(* Schneider Machine Expert - Basic project Grafcet con botonera y flotantes, file version 2.7.0.0 *)
(* ProjectInformations: Name=Nuevo proyecto *)

HARDWARE
  Cpu 0: TM221M16R/G
  ModuleExtensionObject 0: TM3DI16K
  ModuleExtensionObject 1: TM3AI4/G
  EthernetConfiguration: NetworkName=M221, IpAllocationMode=FixedAddress, IpAddress=0.0.0.0, SubnetMask=0.0.0.0
  SerialLineConfiguration: Baud=Baud19200, Parity=ParityEven, DataBits=DataBits8, StopBits=StopBits1, PhysicalMedium=PhysicalMediumRs485, TransmissionMode=TransmissionModeModbusRtu, SlaveId=1, Addressing=SlaveAddressing
  MastTask: UsePeriodScanMode=false, PeriodScan=100
  FastTask: Period=255
  CpuBehavior: StartingMode=StartAsPreviousState, AutoSaveRamOnEeprom=true, WatchdogPeriod=250

SYMBOLS  (address, symbol, comment, settings)
  %M0         "Item detected"
  %M1         "Lid at place"
  %M2         "Base at place"
  %M3         "Part leaving"
  %M4         "Start"
  %M5         "Reset"
  %M6         "Stop"
  %M8         "Auto"
  %M10        "Lids conveyor 1"
  %M11        "Stop blade 1"
  %M13        "Base conveyor 1"
  %M14        "Stop blade 2"
  %M15        "Bases conveyor 2"
  %M16        "Grab"
  %M17        "Start light"
  %M18        "Rest light"
  %M19        "Stop light"
  %M100       "Encendido"
  %X2         "Estado 2"
  %X3         "Estado 3"
  %X5         "Estado 5"
  %X6         "Estado 6"
  %X7         "Estado 7"
  %X8         "Estado 8"
  %X9         "Estado 9"
  %X11        "Estado 11"
  %TM0        "Temporizador estado 11"  [Preset=9, Base=OneSecond]
  %C0         "Contador de piezas finalizadas"  [Preset=1000]

GRAFCET Grafcet Secundario
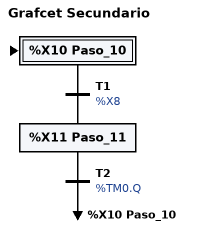
  INITIAL_STEP %X10  (* Paso_10 *)
  STEP %X11  (* Paso_11 *)
  TRANSITION T1 FROM %X10 TO %X11 := %X8;
  TRANSITION T2 FROM %X11 TO %X10 := %TM0.Q;

GRAFCET Grafcet Principal
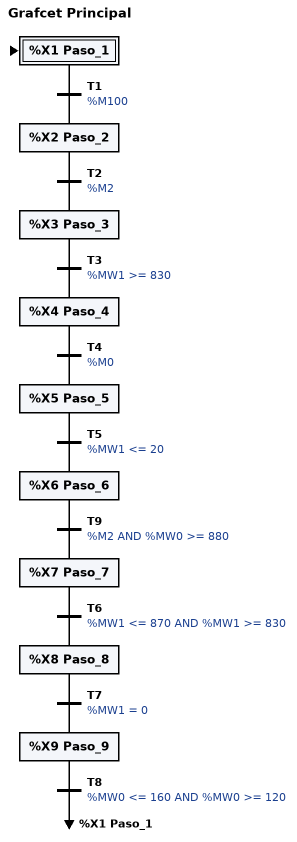
  INITIAL_STEP %X1  (* Paso_1 *)
  STEP %X2  (* Paso_2 *)
  STEP %X3  (* Paso_3 *)
  STEP %X4  (* Paso_4 *)
  STEP %X5  (* Paso_5 *)
  STEP %X6  (* Paso_6 *)
  STEP %X7  (* Paso_7 *)
  STEP %X8  (* Paso_8 *)
  STEP %X9  (* Paso_9 *)
  TRANSITION T1 FROM %X1 TO %X2 := %M100;
  TRANSITION T2 FROM %X2 TO %X3 := %M2;
  TRANSITION T3 FROM %X3 TO %X4 := %MW1 >= 830;
  TRANSITION T4 FROM %X4 TO %X5 := %M0;
  TRANSITION T5 FROM %X5 TO %X6 := %MW1 <= 20;
  TRANSITION T6 FROM %X7 TO %X8 := %MW1 <= 870 AND %MW1 >= 830;
  TRANSITION T7 FROM %X8 TO %X9 := %MW1 = 0;
  TRANSITION T8 FROM %X9 TO %X1 := %MW0 <= 160 AND %MW0 >= 120;
  TRANSITION T9 FROM %X6 TO %X7 := %M2 AND %MW0 >= 880;

TRANSITION T1 (%X10 -> %X11) 
  (* SectionNumber=0 *)

// Rung 0: Tr1
  LD %X8
  ENDT
  // as ST:
  //   TRANSITION := %X8;

TRANSITION T2 (%X11 -> %X10) 
  (* SectionNumber=0 *)

// Rung 1: Tr2
  LD %TM0.Q
  ENDT
  // as ST:
  //   TRANSITION := %TM0.Q;

TRANSITION T1 (%X1 -> %X2) 
  (* SectionNumber=0 *)

// Rung 2: Tr1
  LD %M100
  ENDT
  // as ST:
  //   TRANSITION := %M100;

TRANSITION T2 (%X2 -> %X3) 
  (* SectionNumber=0 *)

// Rung 3: Tr2
  LD %M2
  ENDT
  // as ST:
  //   TRANSITION := %M2;

TRANSITION T3 (%X3 -> %X4) 
  (* SectionNumber=0 *)

// Rung 4: Tr3
  LD [ %MW1 >= 830 ]
  ENDT
  // as ST:
  //   TRANSITION := %MW1 >= 830;

TRANSITION T4 (%X4 -> %X5) 
  (* SectionNumber=0 *)

// Rung 5: Tr4
  LD %M0
  ENDT
  // as ST:
  //   TRANSITION := %M0;

TRANSITION T5 (%X5 -> %X6) 
  (* SectionNumber=0 *)

// Rung 6: Tr5
  LD [ %MW1 <= 20 ]
  ENDT
  // as ST:
  //   TRANSITION := %MW1 <= 20;

TRANSITION T6 (%X7 -> %X8) 
  (* SectionNumber=0 *)

// Rung 7: Tr7
  LD [ %MW1 <= 870 ]
  AND [ %MW1 >= 830 ]
  ENDT
  // as ST:
  //   TRANSITION := %MW1 <= 870 AND %MW1 >= 830;

TRANSITION T7 (%X8 -> %X9) 
  (* SectionNumber=0 *)

// Rung 8: Tr8
  LD [ %MW1 = 0 ]
  ENDT
  // as ST:
  //   TRANSITION := %MW1 = 0;

TRANSITION T8 (%X9 -> %X1) 
  (* SectionNumber=0 *)

// Rung 9: Tr9
  LD [ %MW0 <= 160 ]
  AND [ %MW0 >= 120 ]
  ENDT
  // as ST:
  //   TRANSITION := %MW0 <= 160 AND %MW0 >= 120;

TRANSITION T9 (%X6 -> %X7) 
  (* SectionNumber=0 *)

// Rung 10: Tr6
  LD %M2
  AND [ %MW0 >= 880 ]
  ENDT
  // as ST:
  //   TRANSITION := %M2 AND %MW0 >= 880;

POU Botonera
  (* SectionNumber=13 *)

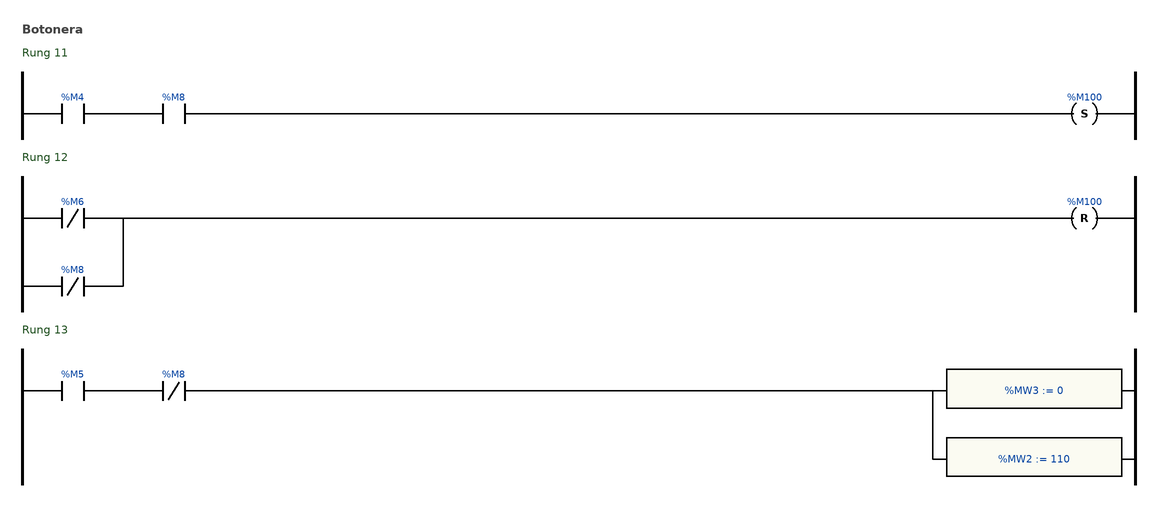

// Rung 11
  LD %M4
  AND %M8
  S %M100
  // as ST:
  //   IF %M4 AND %M8 THEN %M100 := TRUE; END_IF;

// Rung 12
  LDN %M6
  ORN %M8
  R %M100
  // as ST:
  //   IF NOT %M6 OR NOT %M8 THEN %M100 := FALSE; END_IF;

// Rung 13
  LD %M5
  ANDN %M8
  [ %MW3 := 0 ]
  [ %MW2 := 110 ]
  // as ST:
  //   IF %M5 AND NOT %M8 THEN %MW3 := 0; END_IF;
  //   IF %M5 AND NOT %M8 THEN %MW2 := 110; END_IF;

POU Pilotos
  (* SectionNumber=14 *)

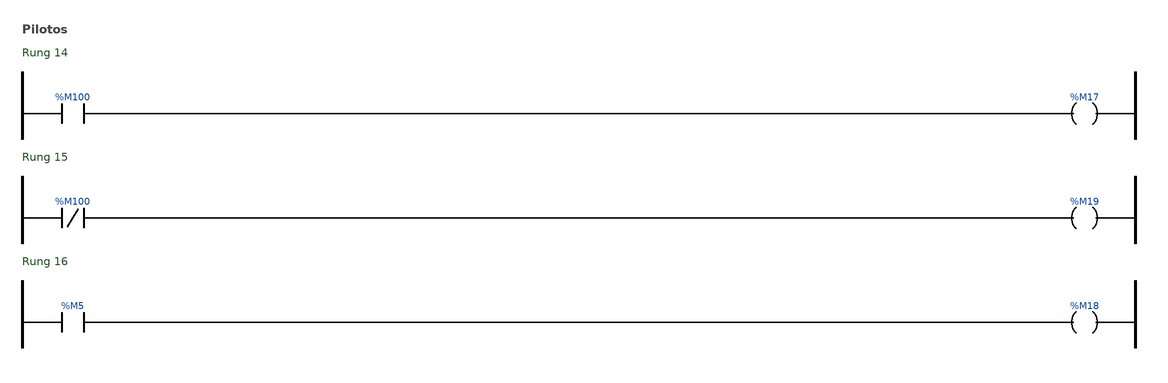

// Rung 14
  LD %M100
  ST %M17
  // as ST:
  //   %M17 := %M100;

// Rung 15
  LDN %M100
  ST %M19
  // as ST:
  //   %M19 := NOT %M100;

// Rung 16
  LD %M5
  ST %M18
  // as ST:
  //   %M18 := %M5;

POU Acciones
  (* SectionNumber=15 *)

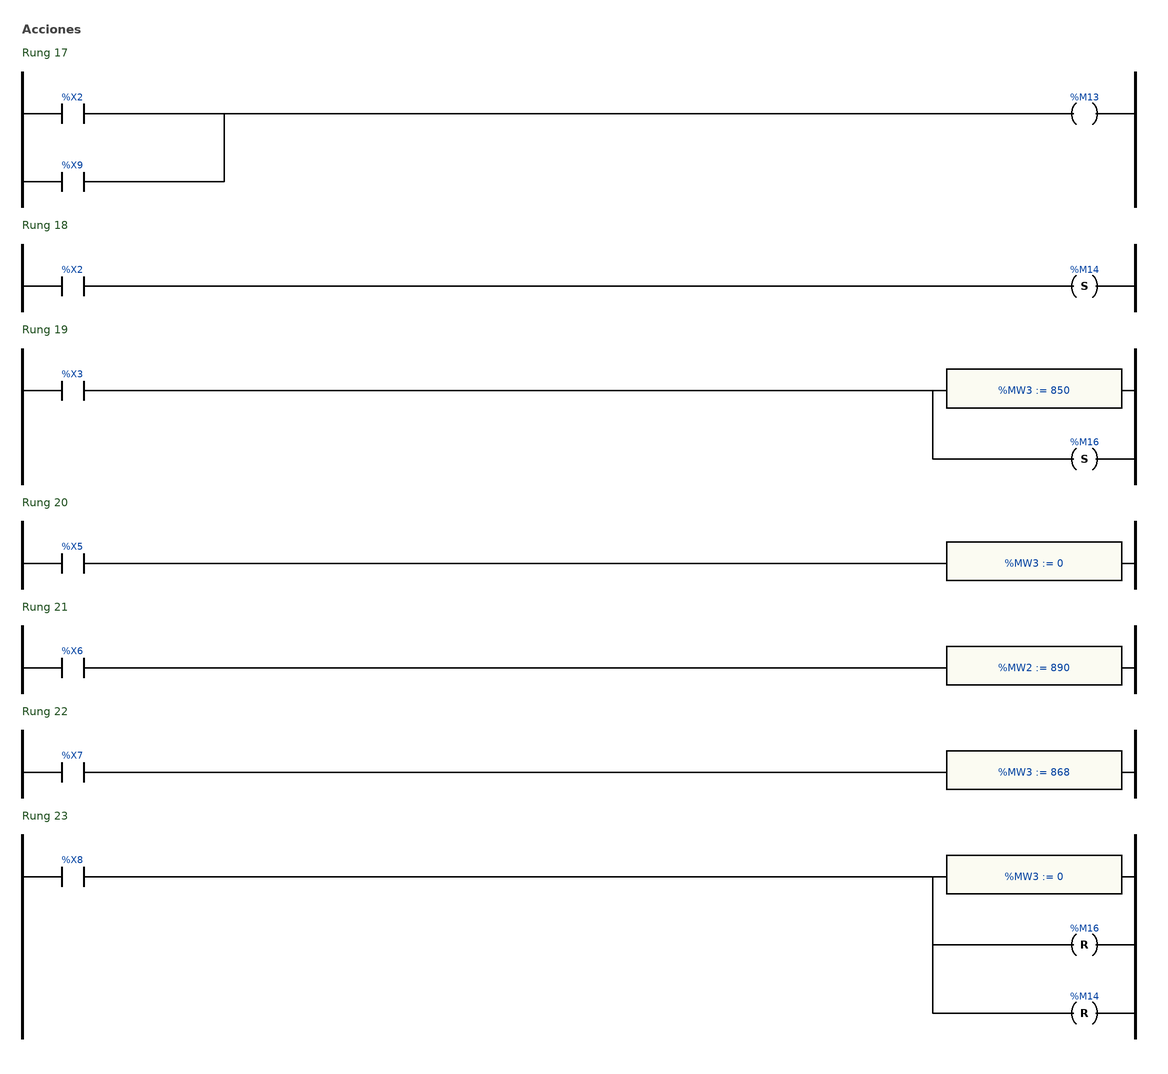

// Rung 17
  LD %X2
  OR %X9
  ST %M13
  // as ST:
  //   %M13 := %X2 OR %X9;

// Rung 18
  LD %X2
  S %M14
  // as ST:
  //   IF %X2 THEN %M14 := TRUE; END_IF;

// Rung 19
  LD %X3
  [ %MW3 := 850 ]
  S %M16
  // as ST:
  //   IF %X3 THEN %MW3 := 850; END_IF;
  //   IF %X3 THEN %M16 := TRUE; END_IF;

// Rung 20
  LD %X5
  [ %MW3 := 0 ]
  // as ST:
  //   IF %X5 THEN %MW3 := 0; END_IF;

// Rung 21
  LD %X6
  [ %MW2 := 890 ]
  // as ST:
  //   IF %X6 THEN %MW2 := 890; END_IF;

// Rung 22
  LD %X7
  [ %MW3 := 868 ]
  // as ST:
  //   IF %X7 THEN %MW3 := 868; END_IF;

// Rung 23
  LD %X8
  [ %MW3 := 0 ]
  R %M16
  R %M14
  // as ST:
  //   IF %X8 THEN %MW3 := 0; END_IF;
  //   IF %X8 THEN %M16 := FALSE; END_IF;
  //   IF %X8 THEN %M14 := FALSE; END_IF;

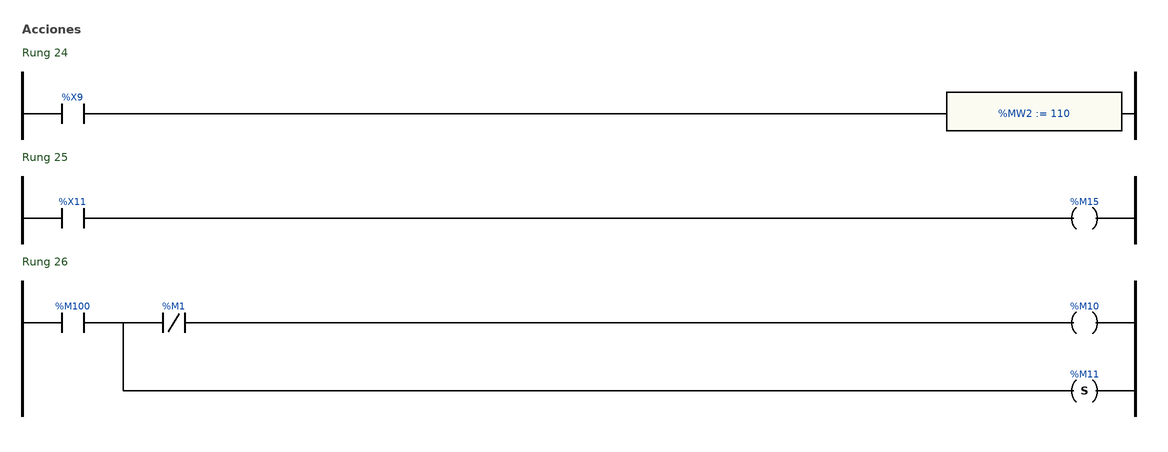

// Rung 24
  LD %X9
  [ %MW2 := 110 ]
  // as ST:
  //   IF %X9 THEN %MW2 := 110; END_IF;

// Rung 25
  LD %X11
  ST %M15
  // as ST:
  //   %M15 := %X11;

// Rung 26
  LD %M100
  MPS
  ANDN %M1
  ST %M10
  MPP
  S %M11
  // as ST:
  //   %M10 := %M100 AND NOT %M1;
  //   IF %M100 THEN %M11 := TRUE; END_IF;

POU Temporizadores y Contadores
  (* SectionNumber=16 *)

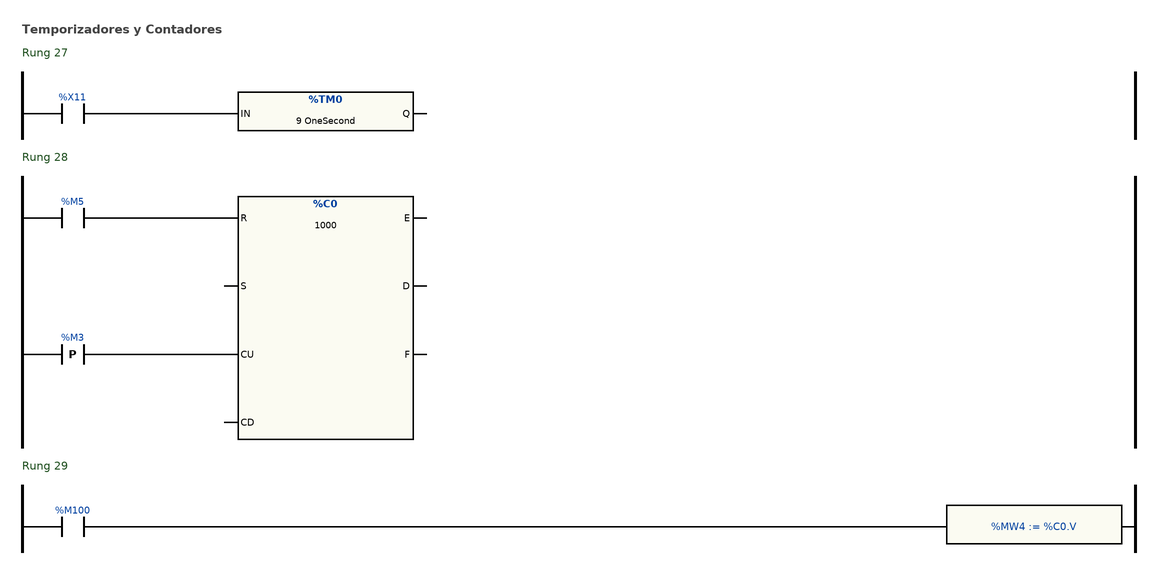

// Rung 27
  BLK %TM0
  LD %X11
  IN
  END_BLK
  // as ST:
  //   %TM0(IN := %X11);

// Rung 28
  BLK %C0
  LD %M5
  R
  LDR %M3
  CU
  END_BLK
  // as ST:
  //   %C0(R := %M5, CU := RISING(%M3));

// Rung 29
  LD %M100
  [ %MW4 := %C0.V ]
  // as ST:
  //   IF %M100 THEN %MW4 := %C0.V; END_IF;
